// TIA Portal V19 export
TYPE "TMeasuringSts"
// stored: Access Published
   STRUCT
      AlarmPresence : Bool;   // Cumulative alarm presence
      InputState : Bool;   // State o input signal of measuring input
      InOperation : Bool;   // Mesuring input in operation
      MeasuringDone_ID : UInt;   // ID of measuring done
      MeasuringValue1 : LReal;   // First measured value
      MeasuringValue2 : LReal;   // Second measured value (for measurement of two edges)
   END_STRUCT;
END_TYPE
